TYPE TFRulliera_OUT :
STRUCT
		FTC_Presenza1 : BOOL;
		FTC_Presenza2 : BOOL;
		FTC_Presenza3 : BOOL;	
		
		
END_STRUCT
END_TYPE

(* stored: Version 1.1.0.1, ProductVersion 3.1.4024.11
   DUT TFRulliera_OUT: Id {d51a01d3-6101-4de6-a428-dcd8cdbf7b26} *)
